Yaskawa INFORM job: TWIN_SKRZYNIA_5140_0_STOPNI_1OBR.JBI

/JOB
//NAME TWIN_SKRZYNIA_5140_0_STOPNI_1OBR
///FOLDERNAME 02-SKRZYNIE_JOBS
//POS
///NPOS 519,519,0,46,4,0
///TOOL 0
///POSTYPE PULSE
///PULSE
C00000=1055,-24125,84372,288,19725,204
C00001=1055,-24125,84372,288,19725,204
C00002=0,-15438,65714,0,-68532,0
C00003=25524,-25821,36823,19654,-58495,38520
C00004=23988,-24960,37134,18595,-57837,38812
C00005=22822,-23954,37534,17811,-57199,39017
C00006=22935,-24057,37491,17887,-57262,38997
C00007=20006,-24258,37408,15644,-56932,39751
C00008=24402,-25289,37013,18874,-58060,38740
C00009=22585,-24665,40358,17164,-59622,30036
C00010=23477,-23257,40205,18030,-58646,29630
C00011=22519,-22398,40568,17384,-58125,29795
C00012=22700,-22567,40495,17506,-58225,29764
C00013=19339,-22794,40398,14955,-57865,30607
C00014=24825,-24328,39798,18931,-59350,29401
C00015=0,-15438,65714,0,-68532,0
C00016=25524,-25821,36823,19654,-58495,38520
C00017=23988,-24960,37134,18595,-57837,38812
C00018=22822,-23954,37534,17811,-57199,39017
C00019=22935,-24057,37491,17887,-57262,38997
C00020=20006,-24258,37408,15644,-56932,39751
C00021=24402,-25289,37013,18874,-58060,38740
C00022=22585,-24665,40358,17164,-59622,30036
C00023=23477,-23257,40205,18030,-58646,29630
C00024=22519,-22398,40568,17384,-58125,29795
C00025=22700,-22567,40495,17506,-58225,29764
C00026=19339,-22794,40398,14955,-57865,30607
C00027=24825,-24328,39798,18931,-59350,29401
C00028=32755,-32613,25711,29640,-48730,33694
C00029=25632,-30899,26166,23992,-46203,35378
C00030=24264,-29862,26497,22996,-45413,35639
C00031=24403,-29974,26459,23097,-45496,35612
C00032=20575,-30233,26374,19602,-44891,36810
C00033=26556,-31526,25988,24663,-46720,35206
C00034=30846,-32795,25752,28021,-48338,30427
C00035=24953,-30697,26306,23444,-45946,31743
C00036=23937,-29910,26558,22702,-45353,31936
C00037=24039,-29993,26530,22778,-45414,31916
C00038=20322,-30240,26449,19379,-44834,33080
C00039=25997,-31433,26093,24205,-46535,31545
C00040=26028,-43665,26580,-39946,8682,24640
C00041=27956,-30595,53065,-101898,6609,54413
C00042=26028,-43663,26580,-39944,8677,24639
C00043=38784,-34544,25404,33956,-51320,34445
C00044=29266,-32676,25756,26732,-47889,36488
C00045=25734,-31262,26119,24020,-46377,37252
C00046=24289,-30200,26441,22967,-45549,37525
C00047=24367,-30262,26420,23025,-45594,37511
C00048=20043,-30544,26331,19080,-44922,38860
C00049=26573,-31816,25967,24631,-46839,37095
C00050=27817,-32566,25782,25532,-47502,36865
C00051=26289,-31635,26016,24424,-46683,37147
C00052=24344,-30243,26427,23007,-45578,37515
C00053=24432,-30312,26405,23072,-45630,37498
C00054=20021,-30599,26315,19050,-44944,38872
C00055=26262,-31616,26021,24405,-46667,37153
C00056=27439,-32346,25835,25259,-47302,36935
C00057=27861,-32554,25785,25570,-47505,36851
C00058=24581,-30384,26384,23190,-45695,37464
C00059=24689,-30466,26358,23269,-45758,37444
C00060=20001,-30771,26264,18999,-45026,38899
C00061=26308,-31607,26026,24448,-46671,37139
C00062=27526,-32360,25834,25329,-47326,36914
C00063=24269,-40076,6479,29767,-34177,34232
C00064=22958,-37632,10123,27061,-35370,35326
C00065=22703,-41294,1722,31272,-29953,33282
C00066=19440,-41515,1663,27208,-29122,34832
C00067=25465,-43501,1200,33269,-31905,32752
C00068=87177,-39066,-1236,81808,-72661,19198
C00069=4794,-34097,38974,4189,-31824,-1302
C00070=4794,-34097,38974,4189,13412,-1302
C00071=11237,-37131,38982,-12694,5333,8253
C00072=6591,-33902,35532,5956,-1761,-1932
C00073=10065,-33530,28876,9373,-31104,-3154
C00074=31877,-32319,25770,29025,-48287,33360
C00075=25178,-31109,26094,23580,-46137,35030
C00076=23652,-29939,26460,22464,-45250,35320
C00077=23742,-30013,26436,22530,-45305,35302
C00078=19630,-30281,26348,18756,-44677,36597
C00079=26056,-31710,25928,24219,-46631,34863
C00080=38095,-40136,7813,41252,-44156,24924
C00081=33231,-38681,8176,37792,-41757,25918
C00082=31538,-37640,8473,36716,-40716,26179
C00083=31687,-37737,8444,36811,-40809,26155
C00084=27389,-38154,8322,32773,-39589,27627
C00085=33834,-39023,8084,38175,-42120,25821
C00086=4801,-35772,25187,4594,-28023,-1125
C00087=-1002,-39861,25115,1795,-37402,-69601
C00088=4264,-34194,25387,4006,-26954,-29436
C00089=4264,-34194,25387,4006,-26954,-81856
C00090=17634,-23800,39238,9573,-31425,-73339
C00091=17837,-27228,32238,10495,-29236,-73805
C00092=17837,-21535,44509,9322,-33342,-73155
C00093=17548,-20734,45666,8935,-33511,-73021
C00094=-20829,-18800,50532,-12466,-37179,-77446
C00095=-20884,-20901,46110,-12960,-35762,-77182
C00096=-20884,-26676,33664,-14451,-31668,-76336
C00097=-20624,-26699,33167,-14265,-31320,-76369
C00098=-33629,-40566,17444,-29603,-33447,-71192
C00099=-33629,-40566,17444,42578,-32312,-84654
C00100=-42160,-31266,16400,42578,-32312,-84654
C00101=-87798,-804,48829,-20188,-26072,-60966
C00102=-76454,-11934,10236,-25964,7954,-64922
C00103=-76448,-11928,10235,-25961,7944,-64914
C00104=-68643,-7759,-23318,-14097,50582,-74897
C00105=-70868,-8793,-8075,-29663,30364,-70765
C00106=-67243,-1968,12282,-49553,26687,-63567
C00107=-68655,-309,14069,-48513,25966,-64203
C00108=-67497,-1678,12591,-49367,26558,-63682
C00109=-71436,-723,2905,-26484,35140,-73726
C00110=-71436,176,6426,-27636,33595,-73066
C00111=-71434,778,8668,-28412,32633,-72624
C00112=-68624,-2689,-85,-28291,36551,-72622
C00113=-99375,3692,5712,40719,48607,-84097
C00114=-94964,4957,10918,40408,44640,-83792
C00115=-93063,6047,12199,39572,43744,-83178
C00116=-94964,4957,10918,40408,44640,-83792
C00117=-94964,5754,13918,41385,43553,-84439
C00118=-94964,4957,10918,40408,44640,-83792
C00119=-90271,-412,-5146,23417,46876,-76529
C00120=-83133,-4088,-8267,6704,41492,-71542
C00121=-83133,-4088,-8267,6704,41492,-71542
C00122=-83133,-4088,-8267,6704,41492,-11598
C00123=-83133,-16026,-8267,6704,41492,-11598
C00124=-83133,-16026,-8267,6704,41492,-11598
C00125=-48225,-19387,30619,3889,32460,-6728
C00126=56943,-39861,25115,1795,-37402,-69601
C00127=29960,-38386,-19607,-115769,-41858,-24264
C00128=65721,-6478,18155,-133323,-22195,3361
C00129=70544,4411,32968,-134868,-18623,4660
C00130=71874,8263,38598,-134556,-17327,4659
C00131=72629,9390,40002,-135279,-16924,5107
C00132=71441,7638,37831,-134139,-17555,4406
C00133=77146,8888,25050,-166574,-32612,18372
C00134=77146,10029,28643,-166204,-31014,18167
C00135=77146,11198,32202,-165803,-29459,17947
C00136=75508,4678,16951,-165715,-35157,17778
C00137=68680,12216,24468,-164340,-40455,-13359
C00138=68362,12845,25743,-164045,-40097,-13561
C00139=68362,13700,28585,-163752,-38808,-13742
C00140=68362,12845,25743,-164045,-40097,-13561
C00141=64993,-1168,28876,-102971,-10760,-49875
C00142=63888,481,30670,-102324,-11438,-50313
C00143=64993,-1168,28876,-102971,-10760,-49875
C00144=58588,-14653,4620,-120782,-19611,-35794
C00145=29960,-38386,-19607,-115769,-41858,-24264
C00146=56943,-39861,25115,1795,-37402,-69601
C00147=-1002,-39861,25115,1795,-37402,-69601
C00148=-1001,-39858,25114,1795,-37402,0
C00149=6591,-33902,35532,5956,-1761,-1932
C00150=6592,-33900,35531,103508,-35512,-26314
C00151=-99253,-13690,44082,59847,13407,-31313
C00152=-85045,-36869,-4353,28502,-22832,-52282
C00153=-92346,-18713,13565,21110,-22545,-55257
C00154=-85370,-14218,16934,32905,-23649,-60330
C00155=-84150,-13282,17685,34842,-23935,-61163
C00156=-82877,-12536,18624,36445,-24482,-61818
C00157=-84150,-13282,17685,34842,-23935,-61163
C00158=-85467,-11480,19558,33086,-23405,-60436
C00159=-84150,-13282,17685,34842,-23935,-61163
C00160=-85732,-21202,11427,30682,-24763,-59235
C00161=-84559,-15616,15722,33768,-24118,-60665
C00162=-84150,-13282,17685,34842,-23935,-61163
C00163=-83260,-12880,18034,36130,-24218,-61709
C00164=-84150,-13282,17685,34842,-23935,-61163
C00165=-85365,-11775,19006,33430,-23307,-60600
C00166=-84150,-13282,17685,34842,-23935,-61163
C00167=-85786,-16909,14677,31743,-23900,-59790
C00168=-84150,-13282,17685,34842,-23935,-61163
C00169=-83215,-12861,18051,36194,-24233,-61735
C00170=-84150,-13282,17685,34842,-23935,-61163
C00171=-85327,-11825,18959,33476,-23327,-60618
C00172=-84150,-13282,17685,34842,-23935,-61163
C00173=-87841,-18519,13420,28367,-23534,-58339
C00174=-84150,-13282,17685,34842,-23935,-61163
C00175=-83292,-12894,18020,36083,-24208,-61688
C00176=-84150,-13282,17685,34842,-23935,-61163
C00177=-85185,-12008,18799,33646,-23400,-60687
C00178=-84150,-13282,17685,34842,-23935,-61163
C00179=-86371,-18277,13606,30568,-23951,-59265
C00180=-84345,-13370,17612,34554,-23873,-61041
C00181=-83240,-12871,18042,36158,-24225,-61720
C00182=-84345,-13370,17612,34554,-23873,-61041
C00183=-85365,-12110,18711,33368,-23345,-60568
C00184=-84345,-13370,17612,34554,-23873,-61041
C00185=-86191,-19647,12567,30467,-24278,-59187
C00186=-84345,-13372,17610,34552,-23873,-61039
C00187=-83096,-12807,18098,36363,-24268,-61804
C00188=-84345,-13372,17610,34552,-23873,-61039
C00189=-85268,-12232,18600,33480,-23393,-60612
C00190=-84345,-13372,17610,34552,-23873,-61039
C00191=-84814,-16043,15376,33312,-24093,-60464
C00192=-84104,-13265,17702,34906,-23948,-61189
C00193=-82960,-12743,18153,36555,-24313,-61887
C00194=-84104,-13265,17702,34906,-23948,-61189
C00195=-84979,-12194,18635,33901,-23496,-60788
C00196=-84104,-13265,17702,34906,-23948,-61189
C00197=-86610,-16845,14732,30573,-23614,-59301
C00198=-84104,-13265,17702,34906,-23948,-61189
C00199=-82793,-12667,18222,36790,-24370,-61986
C00200=-84104,-13265,17702,34906,-23948,-61189
C00201=-84888,-12305,18537,34004,-23540,-60830
C00202=-84104,-13265,17702,34906,-23948,-61189
C00203=-83806,-19585,12613,33764,-25080,-60559
C00204=-83675,-13072,17868,35530,-24083,-61453
C00205=-82553,-12556,18319,37130,-24451,-62127
C00206=-83675,-13072,17868,35530,-24083,-61453
C00207=-84378,-12223,18610,34735,-23716,-61138
C00208=-83675,-13072,17868,35530,-24083,-61453
C00209=-87149,-17993,13826,29513,-23647,-58830
C00210=-84104,-13265,17702,34906,-23948,-61189
C00211=-82640,-12594,18285,37014,-24425,-62079
C00212=-84104,-13265,17702,34906,-23948,-61189
C00213=-84792,-12429,18430,34119,-23592,-60877
C00214=-84104,-13265,17702,34906,-23948,-61189
C00215=-83583,-9185,30892,23668,-36042,-57025
C00216=-85789,-8328,35795,20592,-37093,-55378
C00217=-85786,-16735,14816,31782,-23869,-59812
C00218=-84103,-13263,17702,34906,-23947,-61191
C00219=-83225,-12865,18046,36177,-24227,-61729
C00220=-84103,-13263,17702,34906,-23947,-61191
C00221=-84774,-12447,18412,34138,-23599,-60886
C00222=-84103,-13263,17702,34906,-23947,-61191
C00223=-86149,-16246,6730,18897,-35239,-57128
C00224=-86244,-15289,7532,18875,-35060,-57127
C00225=-85361,-14893,7870,19824,-35193,-57574
C00226=-86244,-15289,7532,18875,-35060,-57127
C00227=-86889,-14409,8282,18264,-34784,-56850
C00228=-86244,-15289,7532,18875,-35060,-57127
C00229=-90262,-21765,2389,14114,-35574,-54847
C00230=-90262,-21765,2389,28730,-17672,-54847
C00231=-89967,-19086,25635,28730,-17672,-54847
C00232=568,-24029,84339,168,19981,112
C00233=568,-24677,83015,164,20405,113
C00234=101153,-24598,83176,165,20353,113
C00235=101153,-24598,83176,165,20353,113
C00236=89967,-19086,25635,-28730,-17672,54847
C00237=90262,-21765,2389,-28730,-17672,54847
C00238=86932,-18662,4771,-17876,-35519,56628
C00239=86578,-15436,7408,-18515,-35011,56957
C00240=85428,-14922,7844,-19753,-35183,57541
C00241=84405,-14447,8250,-20842,-35348,58054
C00242=85428,-14922,7844,-19753,-35183,57541
C00243=86134,-13973,8661,-19091,-34881,57237
C00244=85428,-14922,7844,-19753,-35183,57541
C00245=85786,-16735,14816,-31782,-23869,59812
C00246=83514,-12996,17929,-35760,-24132,61552
C00247=82296,-12429,18424,-37488,-24534,62281
C00248=83514,-12996,17929,-35760,-24132,61552
C00249=84266,-12085,18725,-34910,-23738,61214
C00250=83514,-12996,17929,-35760,-24132,61552
C00251=87323,-6914,39851,-18853,-38149,44508
C00252=83118,-12818,18089,-36330,-24263,61791
C00253=81969,-12276,18566,-37944,-24648,62472
C00254=83118,-12818,18089,-36330,-24263,61791
C00255=83927,-11846,18941,-35423,-23842,61433
C00256=83118,-12818,18089,-36330,-24263,61791
C00257=83806,-19585,12613,-33764,-25080,60559
C00258=83148,-12832,18077,-36287,-24254,61773
C00259=81889,-12236,18598,-38058,-24676,62520
C00260=83148,-12832,18077,-36287,-24254,61773
C00261=83900,-11930,18867,-35446,-23862,61440
C00262=83148,-12832,18077,-36287,-24254,61773
C00263=86610,-16845,14732,-30573,-23614,59301
C00264=82493,-13239,17725,-37070,-24559,62089
C00265=81442,-12739,18159,-38529,-24915,62703
C00266=82493,-13239,17725,-37070,-24559,62089
C00267=83435,-12133,18689,-36040,-24063,61682
C00268=82493,-13239,17725,-37070,-24559,62089
C00269=84814,-16043,15376,-33312,-24093,60464
C00270=82555,-13613,17404,-36910,-24580,62015
C00271=81369,-13053,17885,-38558,-24979,62709
C00272=82555,-13613,17404,-36910,-24580,62015
C00273=83568,-12431,18429,-35805,-24046,61580
C00274=82555,-13613,17404,-36910,-24580,62015
C00275=86191,-19647,12567,-30467,-24278,59187
C00276=82500,-13648,17375,-36975,-24607,62039
C00277=81594,-13224,17740,-38236,-24911,62571
C00278=82500,-13648,17375,-36975,-24607,62039
C00279=83449,-12543,18332,-35941,-24104,61633
C00280=82500,-13648,17375,-36975,-24607,62039
C00281=86371,-18277,13606,-30568,-23951,59265
C00282=82904,-13790,17251,-36416,-24470,61808
C00283=81796,-13275,17692,-37971,-24838,62464
C00284=82904,-13790,17251,-36416,-24470,61808
C00285=83696,-12867,18046,-35547,-24051,61466
C00286=82904,-13790,17251,-36416,-24470,61808
C00287=87841,-18519,13420,-28367,-23534,58339
C00288=82748,-13879,17174,-36603,-24542,61883
C00289=81789,-13434,17554,-37946,-24861,62449
C00290=82748,-13879,17174,-36603,-24542,61883
C00291=83603,-12888,18026,-35668,-24086,61514
C00292=82748,-13879,17174,-36603,-24542,61883
C00293=85786,-16909,14677,-31743,-23900,59790
C00294=82339,-14116,16972,-37087,-24733,62079
C00295=81557,-13752,17280,-38171,-24994,62536
C00296=82339,-14116,16972,-37087,-24733,62079
C00297=83390,-12909,18006,-35951,-24172,61633
C00298=82339,-14116,16972,-37087,-24733,62079
C00299=85732,-21202,11427,-30682,-24763,59235
C00300=82398,-14365,16763,-36952,-24745,62014
C00301=81340,-13876,17176,-38416,-25096,62632
C00302=82398,-14365,16763,-36952,-24745,62014
C00303=83629,-12951,17972,-35620,-24090,61491
C00304=82398,-14365,16763,-36952,-24745,62014
C00305=92346,-18713,13565,-21110,-22545,55257
C00306=82794,-13980,17083,-36511,-24538,61844
C00307=81697,-13472,17516,-38043,-24902,62488
C00308=82794,-13980,17083,-36511,-24538,61844
C00309=83767,-12847,18056,-35444,-24023,61424
C00310=82794,-13980,17083,-36511,-24538,61844
C00311=85045,-36869,-4353,-28502,-22832,52282
C00312=69856,-53931,-13446,-33557,-28911,29591
C00313=73943,-28815,39553,-16801,-45089,19004
C00314=0,-24029,84339,0,19981,0
C00315=0,-24029,84339,0,19981,0
C00316=0,-52280,40443,0,6876,0
C00317=63961,-36661,14391,66570,-58199,13439
C00318=49610,-38907,493,64064,-47684,11073
C00319=46995,-37828,887,63047,-46050,11165
C00320=46896,-37872,871,62973,-46008,11193
C00321=54160,-39955,137,66075,-50361,10746
C00322=0,-52280,40443,0,6876,0
C00323=0,-52280,40443,0,6876,0
C00324=42978,-45587,7631,48214,-41849,18034
C00325=36694,-44945,-1657,49443,-34807,15750
C00326=45692,-38977,-3583,70505,-41697,11397
C00327=45346,-39151,-3505,69979,-41499,11612
C00328=45286,-39124,-3496,69961,-41460,11611
C00329=34756,-41823,-6138,63561,-31389,22119
C00330=59828,-44646,-5405,72855,-48572,12139
C00331=0,-38761,66314,0,-763,0
C00332=0,-44757,54667,0,2744,0
C00333=40382,-38226,12225,48505,-40693,16039
C00334=55481,-27484,23768,62968,-54833,11978
C00335=49932,-26591,24189,59970,-51981,12550
C00336=49523,-31326,12269,55024,-55929,13117
C00337=55330,-33748,11238,57660,-59334,12681
C00338=78664,-24436,10378,82837,-79111,12029
C00339=75189,-23065,11287,81851,-76948,11927
C00340=75189,-45249,11287,81851,-38847,11927
C00341=29880,-45249,11287,43145,-11324,11927
C00342=0,-24029,84339,0,19981,0
C00343=0,-24026,84338,1,19977,2
C00344=4264,-34194,25387,4006,-26954,-29436
C00345=4264,-34194,25387,4006,-26954,-81856
C00346=18580,-28601,30698,11472,-29284,-74138
C00347=-23778,-26243,38799,-16502,-35132,-75964
C00348=18580,-28601,30698,11472,-29284,-74138
C00349=4264,-34194,25387,4006,-26954,-81856
C00350=4264,-34194,25387,4006,-26954,-29436
C00351=1,-24024,84337,2,19973,1
C00352=-64243,-26178,31107,-39513,40312,-5844
C00353=-72148,3973,56008,-35470,42045,-10522
C00354=-72090,16396,76301,-42067,35650,-6519
C00355=-69388,15725,61378,-31740,35177,-8719
C00356=-69127,27099,75569,-32744,34250,-8088
C00357=-67573,2495,11285,-21767,57629,-15193
C00358=-77819,19629,29798,-10454,63174,-20704
C00359=-72990,23583,14304,-10735,77209,-20379
C00360=-74593,38003,46707,-11043,65751,-19814
C00361=-73236,38943,48295,-11400,65557,-19316
C00362=-73329,42107,51779,-6346,67443,-19636
C00363=-87142,34654,46174,17622,63862,-25393
C00364=-87240,36727,48611,18897,66604,-25032
C00365=-99033,21517,12213,24947,79702,-26203
C00366=-91500,-14196,-34781,24472,81625,-22832
C00367=-100472,-45007,-27818,8167,67201,-29302
C00368=0,-36642,16905,0,48372,0
C00369=66009,-61997,-62105,21406,63483,18379
C00370=97242,-23579,-39442,10179,68876,30321
C00371=73684,-7073,-17511,24638,68131,29022
C00372=59136,7235,6676,33270,66602,27507
C00373=54816,14937,6234,39741,69494,31070
C00374=54365,20668,19279,41017,66202,29418
C00375=64503,4223,2857,29650,48528,26647
C00376=75622,3202,-3149,3890,49494,34281
C00377=88036,13177,2413,-18568,66573,35876
C00378=90462,21593,10123,-22613,76266,34479
C00379=92450,29224,20002,-25750,81642,33727
C00380=94949,8131,-12163,-20291,74229,36861
C00381=94949,8084,-13484,-20215,75047,36712
C00382=70412,-34016,-52305,-11724,65624,29757
C00383=44268,-30306,-1568,-7370,48673,18708
C00384=1,-24024,84337,2,19973,1
C00385=1,-24024,84337,2,19973,1
C00386=3796,-57671,22373,2336,-25309,-753
C00387=52632,-34554,16626,51161,-63050,5622
C00388=59461,-32779,9832,66317,-58406,17312
C00389=52359,-27861,19114,60105,-56373,14901
C00390=51089,-17517,41583,51411,-64544,19432
C00391=62932,-33588,12189,66848,-61063,18031
C00392=55769,-31640,17107,64026,-54372,11197
C00393=49968,-26926,23568,59773,-52215,12586
C00394=49609,-31413,12230,55051,-55993,13121
C00395=55330,-33748,11238,57660,-59334,12681
C00396=62932,-33588,12189,66848,-61063,18031
C00397=1,-24024,84337,2,19973,1
C00398=1,-24024,84337,2,19973,1
C00399=57188,-41777,19973,48132,-58706,4905
C00400=55566,-48748,-16991,79805,-45048,-6941
C00401=49908,-48716,-25784,90749,-41340,-3650
C00402=44463,-47168,-25441,90895,-37884,-4475
C00403=44064,-46950,-25361,90973,-37634,-4568
C00404=55479,-50244,-26473,91085,-44870,-3042
C00405=12119,-24859,71505,13236,4440,2633
C00406=-91085,-34291,10385,1908,-24348,-42097
C00407=-86191,-19647,12567,30467,-24278,-59187
C00408=-99260,-11699,19072,-14181,-20214,-40097
C00409=-98334,-11556,19569,-10380,-20328,-41527
C00410=-99474,-20389,12397,-11593,-22150,-41069
C00411=0,-52280,40443,0,6876,0
C00412=85348,-24204,23536,-13963,-15515,44275
C00413=84670,-17015,14597,-33277,-24304,60423
C00414=97099,-12623,18260,8611,-19973,42508
C00415=97182,-12918,18001,8747,-20027,42449
C00416=96230,-24528,9149,6144,-22576,43630
C00417=0,-52280,40443,0,6876,0
C00418=0,-52280,40443,0,6876,0
C00419=-90140,-60305,18108,-2708,1721,-7625
C00420=-95594,-27428,6866,-4663,-19832,-42154
C00421=-99356,-13410,18355,-15385,-17730,-37479
C00422=-99405,-10878,20508,-15853,-17333,-37255
C00423=-99155,-10757,20617,-15328,-17277,-37477
C00424=-99152,-3438,39174,-10973,-24351,-39660
C00425=-99136,-3399,39184,-10956,-24327,-39665
C00426=-100183,-18601,14070,-16273,-18800,-37146
C00427=-90140,-60305,18108,-2708,1721,-7625
C00428=0,-52280,40443,0,6876,0
C00429=84259,-57935,27522,-3761,3673,6310
C00430=86507,-39672,4297,-27618,-16640,46340
C00431=70477,-27878,7073,-45786,-32339,64941
C00432=84043,-16293,15174,-34312,-24409,60872
C00433=82317,-21832,-7005,-55296,-17985,71248
C00434=99154,-17369,4403,32227,-9753,28926
C00435=99154,-17369,4403,32227,-9753,28926
C00436=98946,-17182,4556,31649,-9649,29182
C00437=100388,-17987,13832,15751,-21517,39479
C00438=86507,-39672,4297,-27618,-16640,46340
C00439=84259,-57935,27522,-3761,3673,6310
C00440=0,-52280,40443,0,6876,0
C00441=0,-27933,77061,0,20812,0
C00442=0,-27933,77061,0,20812,0
C00443=0,-52280,40443,0,6876,0
C00444=-91970,-60791,14435,-3343,512,-9412
C00445=-99196,-15868,16098,-13748,-19297,-38710
C00446=-99196,-15868,16098,-13748,-19297,-38710
C00447=-99196,-15868,16098,-13748,-19297,-38710
C00448=-85815,-11758,19597,31748,-21097,-58265
C00449=-87383,-11883,19487,26986,-20206,-56250
C00450=-99562,-16264,15781,-14410,-19427,-38431
C00451=-99196,-15868,16098,-13748,-19297,-38710
C00452=-91970,-60791,14435,-3343,512,-9412
C00453=0,-52280,40443,0,6876,0
C00454=91083,-60784,14823,-9043,-825,15173
C00455=83869,-19403,12921,-33769,-24740,60260
C00456=83869,-19403,12921,-33769,-24740,60260
C00457=83420,-14897,16486,-35538,-24144,61113
C00458=90568,-11796,19695,-13982,-20788,51525
C00459=90396,-11649,19890,-14205,-20868,51587
C00460=95871,-14889,15992,4901,-19605,43825
C00461=83869,-19403,12921,-33769,-24740,60260
C00462=91083,-60784,14823,-9043,-825,15173
C00463=0,-52280,40443,0,6876,0
C00464=-91526,-60598,16699,7584,176,-13289
C00465=-94392,-6553,48683,5805,-47321,-49764
C00466=-88951,-345,54953,10686,-47392,-51569
C00467=-88172,5833,62122,11322,-47753,-51785
C00468=-90970,-13982,9528,8812,-34392,-51924
C00469=-84917,-15593,15742,33275,-23984,-60461
C00470=-81669,-15982,15425,37506,-25258,-62202
C00471=-79867,-25377,9541,37586,-25936,-59971
C00472=-91415,-60262,16631,7870,-73,-13734
C00473=24,-24029,84339,7,19981,5
C00474=160,-24029,84339,47,19981,32
C00475=99096,-24029,84339,47,19981,32
C00476=99096,-24029,84339,47,19981,32
C00477=89967,-19086,25635,-28730,-17672,54847
C00478=85786,-16735,14816,-31782,-23869,59812
C00479=83492,-14473,16674,-35480,-24338,61406
C00480=82750,-11489,19288,-37313,-24360,62208
C00481=85452,-13705,8809,-19525,-34825,57501
C00482=85505,-16299,6686,-19564,-35388,57437
C00483=89967,-19086,25635,-28730,-17672,54847
C00484=568,-24029,84339,168,19981,112
C00485=568,-24029,84339,168,19981,112
C00486=-91970,-60791,14435,-3343,512,-9412
C00487=-86948,-23217,10819,28314,-23349,-56438
C00488=-85895,-16522,15767,31843,-22281,-58087
C00489=-93602,1725,52992,2981,-38211,-34794
C00490=-93409,-737,47229,3345,-36106,-34967
C00491=-86145,-24679,9854,29028,-23971,-56682
C00492=-100471,-58311,4157,14142,-4822,-27614
C00493=-68517,-58311,4157,14142,-4822,-27614
C00494=0,-52280,40443,0,6876,0
C00495=91083,-60784,14823,-9043,-825,15173
C00496=83869,-19403,12921,-33769,-24740,60260
C00497=82620,-18743,14708,-32942,-26226,58979
C00498=83365,-11429,20745,-33501,-24845,59379
C00499=83361,-11160,20982,-33549,-24816,59402
C00500=84798,-22668,11879,-29033,-26372,57255
C00501=91083,-60784,14823,-9043,-825,15173
C00502=0,-52280,40443,0,6876,0
C00503=-6369,-39206,65423,-4801,-482,2563
C00504=-97287,-29142,12714,-8673,-22288,-37832
C00505=-86191,-19647,12567,30467,-24278,-59187
C00506=-85671,-16302,15857,30808,-24404,-58999
C00507=-100033,-10430,22389,-14713,-22552,-38787
C00508=-95758,-10871,21797,-1120,-21702,-44724
C00509=-87910,-17792,15835,25414,-24996,-56048
C00510=-97287,-29142,12714,-8673,-22288,-37832
C00511=0,-52280,40443,0,6876,0
C00512=92301,-25634,22749,2368,-15645,37646
C00513=83738,-18329,13570,-34202,-24868,60772
C00514=90096,-13099,18146,-15422,-20883,52700
C00515=93330,-13245,17928,-4627,-20146,48105
C00516=80226,-20465,12178,-39626,-27411,62762
C00517=92301,-25634,22749,2368,-15645,37646
C00518=0,-52280,40443,0,6876,0
BC00000=413138
BC00001=413138
BC00002=413138
BC00003=290246
BC00004=290246
BC00005=290246
BC00006=290246
BC00007=290246
BC00008=290246
BC00009=347127
BC00010=347132
BC00011=347132
BC00012=347132
BC00013=347132
BC00014=347132
BC00015=413138
BC00016=413134
BC00017=413134
BC00018=413134
BC00019=413134
BC00020=413134
BC00021=413134
BC00022=474623
BC00023=474628
BC00024=474628
BC00025=474628
BC00026=474628
BC00027=474628
BC00028=522849
BC00029=522849
BC00030=522849
BC00031=522849
BC00032=522849
BC00033=522849
BC00034=586045
BC00035=586045
BC00036=586045
BC00037=586045
BC00038=586045
BC00039=586045
BC00040=479622
BC00041=618860
BC00042=673957
BC00043=655410
BC00044=655410
BC00045=655410
BC00046=655410
BC00047=655410
BC00048=655410
BC00049=655410
BC00050=708270
BC00051=708270
BC00052=708270
BC00053=708270
BC00054=708270
BC00055=708270
BC00056=770184
BC00057=770184
BC00058=770184
BC00059=770184
BC00060=770184
BC00061=770184
BC00062=823730
BC00063=829967
BC00064=829969
BC00065=829970
BC00066=829970
BC00067=829970
BC00068=838761
BC00069=740349
BC00070=687700
BC00071=771943
BC00072=861898
BC00073=881669
BC00074=901229
BC00075=901229
BC00076=901229
BC00077=901229
BC00078=901229
BC00079=901229
BC00080=949836
BC00081=949836
BC00082=949836
BC00083=949836
BC00084=949836
BC00085=949836
BC00086=922151
BC00087=915598
BC00088=911152
BC00089=906014
BC00090=926513
BC00091=926513
BC00092=930959
BC00093=930959
BC00094=930959
BC00095=930959
BC00096=930959
BC00097=930959
BC00098=930959
BC00099=930959
BC00100=930959
BC00101=930959
BC00102=930959
BC00103=948711
BC00104=959797
BC00105=976501
BC00106=976501
BC00107=976501
BC00108=976501
BC00109=976501
BC00110=976501
BC00111=976502
BC00112=976502
BC00113=976502
BC00114=976502
BC00115=976502
BC00116=976502
BC00117=976502
BC00118=976502
BC00119=966879
BC00120=952245
BC00121=926980
BC00122=926980
BC00123=926980
BC00124=893798
BC00125=874726
BC00126=930959
BC00127=930959
BC00128=930959
BC00129=947173
BC00130=952334
BC00131=952334
BC00132=952334
BC00133=952334
BC00134=952334
BC00135=952334
BC00136=952334
BC00137=952334
BC00138=952334
BC00139=952334
BC00140=952334
BC00141=952334
BC00142=952334
BC00143=952334
BC00144=946821
BC00145=930959
BC00146=900237
BC00147=900237
BC00148=930961
BC00149=861898
BC00150=861901
BC00151=861901
BC00152=931504
BC00153=960562
BC00154=960559
BC00155=960559
BC00156=960559
BC00157=960559
BC00158=960559
BC00159=960559
BC00160=902188
BC00161=902188
BC00162=902188
BC00163=902188
BC00164=902188
BC00165=902188
BC00166=902188
BC00167=840744
BC00168=840744
BC00169=840744
BC00170=840744
BC00171=840744
BC00172=840744
BC00173=779300
BC00174=779300
BC00175=779300
BC00176=779300
BC00177=779300
BC00178=779300
BC00179=717855
BC00180=717855
BC00181=717855
BC00182=717855
BC00183=717855
BC00184=717855
BC00185=656405
BC00186=656405
BC00187=656405
BC00188=656405
BC00189=656405
BC00190=656405
BC00191=594961
BC00192=594961
BC00193=594961
BC00194=594961
BC00195=594961
BC00196=594961
BC00197=533517
BC00198=533517
BC00199=533517
BC00200=533517
BC00201=533517
BC00202=533517
BC00203=472073
BC00204=472073
BC00205=472073
BC00206=472073
BC00207=472073
BC00208=472073
BC00209=410629
BC00210=410629
BC00211=410629
BC00212=410629
BC00213=410629
BC00214=410629
BC00215=410629
BC00216=349186
BC00217=349186
BC00218=349186
BC00219=349186
BC00220=349186
BC00221=349186
BC00222=349186
BC00223=336469
BC00224=336469
BC00225=336469
BC00226=336469
BC00227=336469
BC00228=336469
BC00229=336469
BC00230=336469
BC00231=336469
BC00232=336469
BC00233=511557
BC00234=512005
BC00235=363797
BC00236=336469
BC00237=336469
BC00238=337415
BC00239=337415
BC00240=337415
BC00241=337415
BC00242=337415
BC00243=337415
BC00244=337415
BC00245=349186
BC00246=350137
BC00247=350137
BC00248=350137
BC00249=350137
BC00250=350137
BC00251=410629
BC00252=411580
BC00253=411580
BC00254=411580
BC00255=411580
BC00256=411580
BC00257=472073
BC00258=473025
BC00259=473025
BC00260=473025
BC00261=473025
BC00262=473025
BC00263=533517
BC00264=534468
BC00265=534468
BC00266=534468
BC00267=534468
BC00268=534468
BC00269=594961
BC00270=594961
BC00271=594961
BC00272=594961
BC00273=594961
BC00274=594961
BC00275=656405
BC00276=657350
BC00277=657350
BC00278=657350
BC00279=657350
BC00280=657350
BC00281=717855
BC00282=718799
BC00283=718799
BC00284=718799
BC00285=718799
BC00286=718799
BC00287=779300
BC00288=780245
BC00289=780245
BC00290=780245
BC00291=780245
BC00292=780245
BC00293=840744
BC00294=841691
BC00295=841691
BC00296=841691
BC00297=841691
BC00298=841691
BC00299=902188
BC00300=903136
BC00301=903136
BC00302=903136
BC00303=903136
BC00304=903136
BC00305=963634
BC00306=963633
BC00307=963633
BC00308=963633
BC00309=963633
BC00310=963633
BC00311=931504
BC00312=861901
BC00313=861901
BC00314=769966
BC00315=769966
BC00316=716865
BC00317=660977
BC00318=660977
BC00319=660977
BC00320=717171
BC00321=717171
BC00322=716865
BC00323=796033
BC00324=895097
BC00325=895097
BC00326=895097
BC00327=945882
BC00328=959029
BC00329=966042
BC00330=945882
BC00331=840120
BC00332=538973
BC00333=485226
BC00334=456696
BC00335=456696
BC00336=417276
BC00337=417276
BC00338=493986
BC00339=514306
BC00340=514306
BC00341=514306
BC00342=493986
BC00343=797003
BC00344=895791
BC00345=895791
BC00346=895791
BC00347=900237
BC00348=895791
BC00349=895791
BC00350=895791
BC00351=797001
BC00352=812363
BC00353=812363
BC00354=853712
BC00355=873598
BC00356=898537
BC00357=930469
BC00358=930469
BC00359=957978
BC00360=957978
BC00361=957978
BC00362=957979
BC00363=957979
BC00364=957980
BC00365=957980
BC00366=957980
BC00367=872638
BC00368=831236
BC00369=914776
BC00370=953896
BC00371=953897
BC00372=953897
BC00373=984144
BC00374=984144
BC00375=984144
BC00376=984144
BC00377=984144
BC00378=984147
BC00379=984147
BC00380=984147
BC00381=957741
BC00382=957741
BC00383=888928
BC00384=797001
BC00385=461290
BC00386=507200
BC00387=551170
BC00388=578587
BC00389=593948
BC00390=529848
BC00391=529848
BC00392=333808
BC00393=332068
BC00394=295166
BC00395=294388
BC00396=529848
BC00397=461290
BC00398=663315
BC00399=778314
BC00400=778312
BC00401=778312
BC00402=778312
BC00403=838222
BC00404=838222
BC00405=566410
BC00406=679663
BC00407=656405
BC00408=656405
BC00409=717855
BC00410=717855
BC00411=717855
BC00412=662303
BC00413=657350
BC00414=657350
BC00415=718803
BC00416=718803
BC00417=717855
BC00418=792672
BC00419=792672
BC00420=896850
BC00421=895720
BC00422=895720
BC00423=957178
BC00424=957178
BC00425=959216
BC00426=957178
BC00427=792672
BC00428=792672
BC00429=792672
BC00430=887446
BC00431=903126
BC00432=903126
BC00433=923336
BC00434=964577
BC00435=976097
BC00436=978451
BC00437=964577
BC00438=887446
BC00439=792672
BC00440=792672
BC00441=700249
BC00442=546214
BC00443=546214
BC00444=546211
BC00445=546211
BC00446=406776
BC00447=406776
BC00448=406778
BC00449=468200
BC00450=468200
BC00451=546211
BC00452=546211
BC00453=546214
BC00454=546214
BC00455=507604
BC00456=410782
BC00457=410782
BC00458=410782
BC00459=472720
BC00460=472720
BC00461=507604
BC00462=546214
BC00463=546214
BC00464=516757
BC00465=383716
BC00466=349186
BC00467=349186
BC00468=336469
BC00469=349186
BC00470=410629
BC00471=416512
BC00472=515801
BC00473=520018
BC00474=474013
BC00475=474013
BC00476=403108
BC00477=336469
BC00478=349186
BC00479=349186
BC00480=349186
BC00481=337415
BC00482=337415
BC00483=336469
BC00484=336469
BC00485=428401
BC00486=546211
BC00487=591088
BC00488=591088
BC00489=591088
BC00490=531116
BC00491=529640
BC00492=529640
BC00493=529640
BC00494=529640
BC00495=546214
BC00496=589919
BC00497=595627
BC00498=595627
BC00499=534177
BC00500=534177
BC00501=546214
BC00502=529640
BC00503=651195
BC00504=765890
BC00505=777968
BC00506=778453
BC00507=779252
BC00508=840748
BC00509=840748
BC00510=765890
BC00511=717855
BC00512=741100
BC00513=780224
BC00514=780222
BC00515=841743
BC00516=841743
BC00517=741100
BC00518=717855
///POSTYPE BASE
///RECTAN
///RCONF 1,0,0,0,0,0,0,0,0,0,0,0,0,0,0,0,0,0,0,0,0,0,0,0
P00006=0.000,0.000,0.000,0.0000,0.0000,0.0000
P00098=-0.089,-2.467,4.059,0.0000,0.0000,0.0000
P00099=0.011,-2.380,1.226,0.0000,0.0000,0.0000
P00100=-0.081,2.558,4.482,0.0000,0.0000,0.0000
P00101=0.030,-2.286,2.993,0.0000,0.0000,0.0000
P00102=-0.005,-1.108,1.644,0.0000,0.0000,0.0000
P00103=-0.094,-3.400,4.200,0.0000,0.0000,0.0000
P00104=0.043,-2.127,5.826,0.0000,0.0000,0.0000
P00105=-0.043,0.662,5.286,0.0000,0.0000,0.0000
P00106=-0.018,-2.519,0.237,0.0000,0.0000,0.0000
P00107=-0.008,-4.537,-4.500,0.0000,0.0000,0.0000
P00108=0.014,-3.040,2.637,0.0000,0.0000,0.0000
P00109=0.017,-3.622,2.341,0.0000,0.0000,0.0000
P00110=7346.140,158.997,-946.107,-0.1876,37.7131,-155.1643
P00111=7345.905,-141.160,-945.062,8.1413,34.2244,-174.1788
P00112=7393.287,158.977,-939.640,-0.1938,37.7128,-155.1905
P00113=7393.259,-141.170,-939.228,8.1507,34.2195,-174.1496
///RCONF 0,0,0,0,0,0,0,0,0,0,0,0,0,0,0,0,0,0,0,0,0,0,0,0
P00280=-0.761,-1.221,0.004,0.0000,0.0000,0.0000
///RCONF 1,0,0,0,0,0,0,0,0,0,0,0,0,0,0,0,0,0,0,0,0,0,0,0
P00281=-0.866,-3.587,-0.008,0.0000,0.0000,0.0000
///RCONF 0,0,0,0,1,0,0,0,0,0,0,0,0,0,0,0,0,0,0,0,0,0,0,0
P00290=-0.023,-0.050,5.560,0.0000,0.0000,0.0000
///RCONF 1,0,0,0,0,0,0,0,0,0,0,0,0,0,0,0,0,0,0,0,0,0,0,0
P00291=0.002,-0.893,4.526,0.0000,0.0000,0.0000
P00300=-0.036,-1.505,2.318,0.0000,0.0000,0.0000
P00301=0.046,-2.112,7.779,0.0000,0.0000,0.0000
P00302=-0.180,-2.409,6.326,0.0000,0.0000,0.0000
///RCONF 0,0,0,0,0,0,0,0,0,0,0,0,0,0,0,0,0,0,0,0,0,0,0,0
P00303=-0.004,-1.437,-4.584,0.0000,0.0000,0.0000
P00304=0.028,-1.666,-4.234,0.0000,0.0000,0.0000
P00305=-0.003,-1.920,-3.501,0.0000,0.0000,0.0000
P00306=0.015,-2.252,-3.054,0.0000,0.0000,0.0000
P00307=0.019,-2.151,-5.077,0.0000,0.0000,0.0000
P00308=-0.003,-2.092,-4.888,0.0000,0.0000,0.0000
P00309=-0.040,-2.205,-4.992,0.0000,0.0000,0.0000
P00310=-0.006,-2.490,-5.925,0.0000,0.0000,0.0000
P00311=-0.007,-2.079,-5.307,0.0000,0.0000,0.0000
P00350=11.519,-0.008,1.149,0.0000,0.0000,0.0000
P00351=13.563,-0.027,-0.653,0.0000,0.0000,0.0000
P00352=13.252,-0.027,-0.827,0.0000,0.0000,0.0000
P00353=10.971,-0.082,0.776,0.0000,0.0000,0.0000
P00354=-0.024,2.508,-1.824,0.0000,0.0000,0.0000
P00355=-0.001,2.528,-1.131,0.0000,0.0000,0.0000
P00356=-0.034,2.921,-0.262,0.0000,0.0000,0.0000
P00357=0.003,3.386,-0.091,0.0000,0.0000,0.0000
P00358=0.014,3.037,-0.020,0.0000,0.0000,0.0000
P00359=-0.005,2.731,0.912,0.0000,0.0000,0.0000
P00360=-0.011,3.412,0.438,0.0000,0.0000,0.0000
P00361=0.018,3.050,1.253,0.0000,0.0000,0.0000
P00777=-1.000,0.000,-1.000,0.0000,0.0000,0.0000
BP00110=5931.608
BP00111=5960.552
BP00112=5960.545
BP00113=5960.552
//INST
///DATE 2024/12/18 10:28
///ATTR SC,RW
///GROUP1 RB1,BS1
NOP
CALL JOB:MOVE_INTO_TUNNEL
MOVJ C00000 BC00000 VJ=30.00
'------------------------
'------------------------
'SPOINA SRODEK DOL
'------------------------
'------------------------
'POMIAR DO WYJ!! PRZEROBIC NA STD
MOVJ C00001 BC00001 VJ=40.00
MOVJ C00002 BC00002 VJ=40.00
'SPOINA_PODLOGA_BRAK_ROZP
MOVJ C00003 BC00003 VJ=20.00 PL=0
MOVL C00004 BC00004 V=166.7 PL=0
REFP 3 C00005 BC00005
CALL JOB:SEARCH-R1
SET P0098 P0006
SFTON P0098
MOVL C00006 BC00006 V=66.7 PL=0
REFP 3 C00007 BC00007
CALL JOB:SEARCH-R1
SET P0098 P0006
SFTON P0098
MOVL C00008 BC00008 V=333.3 PL=0
SFTOF
'W3L
MOVL C00009 BC00009 V=666.7
MOVL C00010 BC00010 V=166.7 PL=0
REFP 3 C00011 BC00011
CALL JOB:SEARCH-R1
SET P0099 P0006
SFTON P0099
MOVL C00012 BC00012 V=166.7 PL=0
REFP 3 C00013 BC00013
CALL JOB:SEARCH-R1
SET P0099 P0006
SFTON P0099
MOVL C00014 BC00014 V=333.3 PL=0
SFTOF
'SPOINA_PODLOGA_BRAK_ROZP
MOVJ C00015 BC00015 VJ=40.00
'W3P
MOVJ C00016 BC00016 VJ=20.00 PL=0
MOVL C00017 BC00017 V=166.7 PL=0
REFP 3 C00018 BC00018
CALL JOB:SEARCH-R1
SET P0100 P0006
SFTON P0100
MOVL C00019 BC00019 V=66.7 PL=0
REFP 3 C00020 BC00020
CALL JOB:SEARCH-R1
SET P0100 P0006
SFTON P0100
MOVL C00021 BC00021 V=333.3 PL=0
SFTOF
'W3L
MOVL C00022 BC00022 V=666.7
MOVL C00023 BC00023 V=166.7 PL=0
REFP 3 C00024 BC00024
CALL JOB:SEARCH-R1
SET P0101 P0006
SFTON P0101
MOVL C00025 BC00025 V=166.7 PL=0
REFP 3 C00026 BC00026
CALL JOB:SEARCH-R1
SET P0101 P0006
SFTON P0101
MOVL C00027 BC00027 V=333.3 PL=0
SFTOF
'W9P
MOVL C00028 BC00028 V=666.7
MOVL C00029 BC00029 V=166.7
REFP 3 C00030 BC00030
CALL JOB:SEARCH-R1
SET P0102 P0006
SFTON P0102
MOVL C00031 BC00031 V=166.7 PL=0
REFP 3 C00032 BC00032
CALL JOB:SEARCH-R1
SET P0102 P0006
SFTON P0102
MOVL C00033 BC00033 V=333.3 PL=0
'W9L
MOVL C00034 BC00034 V=666.7
MOVL C00035 BC00035 V=166.7
REFP 3 C00036 BC00036
CALL JOB:SEARCH-R1
SET P0103 P0006
SFTON P0103
MOVL C00037 BC00037 V=166.7 PL=0
REFP 3 C00038 BC00038
CALL JOB:SEARCH-R1
SET P0103 P0006
SFTON P0103
MOVL C00039 BC00039 V=333.3 PL=0
'PRZEJAZ NAD BELKA
MOVL C00040 BC00040 V=666.7
MOVJ C00041 BC00041 VJ=40.00
MOVJ C00042 BC00042 VJ=40.00
MOVJ C00043 BC00043 VJ=40.00
'W1P
MOVJ C00044 BC00044 VJ=20.00 PL=0
MOVL C00045 BC00045 V=166.7 PL=0
REFP 3 C00046 BC00046
CALL JOB:SEARCH-R1
SET P0104 P0006
SFTON P0104
MOVL C00047 BC00047 V=166.7 PL=0
REFP 3 C00048 BC00048
CALL JOB:SEARCH-R1
SET P0104 P0006
SFTON P0104
MOVL C00049 BC00049 V=333.3 PL=0
SFTOF
'W1L
MOVL C00050 BC00050 V=666.7
MOVL C00051 BC00051 V=166.7 PL=0
REFP 3 C00052 BC00052
CALL JOB:SEARCH-R1
SET P0105 P0006
SFTON P0105
MOVL C00053 BC00053 V=166.7 PL=0
REFP 3 C00054 BC00054
CALL JOB:SEARCH-R1
SET P0105 P0006
SFTON P0105
MOVL C00055 BC00055 V=333.3 PL=0
SFTOF
MOVL C00056 BC00056 V=666.7
'W10P
MOVL C00057 BC00057 V=166.7 PL=0
REFP 3 C00058 BC00058
CALL JOB:SEARCH-R1
SET P0106 P0006
SFTON P0106
MOVL C00059 BC00059 V=166.7 PL=0
REFP 3 C00060 BC00060
CALL JOB:SEARCH-R1
SET P0106 P0006
SFTON P0106
MOVL C00061 BC00061 V=333.3 PL=0
SFTOF
'W10L
MOVL C00062 BC00062 V=333.3
MOVL C00063 BC00063 V=166.7 PL=0
REFP 3 C00064 BC00064
CALL JOB:SEARCH-R1
SET P0107 P0006
SFTON P0107
MOVL C00065 BC00065 V=166.7 PL=0
REFP 3 C00066 BC00066
CALL JOB:SEARCH-R1
SET P0107 P0006
SFTON P0107
MOVL C00067 BC00067 V=333.3 PL=0
SFTOF
MOVL C00068 BC00068 V=333.3
'PRZEJAZD
MOVJ C00069 BC00069 VJ=50.00
MOVJ C00070 BC00070 VJ=50.00
MOVJ C00071 BC00071 VJ=60.00
MOVJ C00072 BC00072 VJ=60.00
MOVJ C00073 BC00073 VJ=60.00
MOVJ C00074 BC00074 VJ=60.00 PL=0
MOVL C00075 BC00075 V=166.7 PL=0
REFP 3 C00076 BC00076
CALL JOB:SEARCH-R1
SET P0108 P0006
SFTON P0108
MOVL C00077 BC00077 V=166.7 PL=0
REFP 3 C00078 BC00078
CALL JOB:SEARCH-R1
SET P0108 P0006
SFTON P0108
MOVL C00079 BC00079 V=333.3 PL=0
SFTOF
'W2P
'W2L
MOVL C00080 BC00080 V=666.7
MOVL C00081 BC00081 V=166.7 PL=0
REFP 3 C00082 BC00082
CALL JOB:SEARCH-R1
SET P0109 P0006
SFTON P0109
MOVL C00083 BC00083 V=166.7 PL=0
REFP 3 C00084 BC00084
CALL JOB:SEARCH-R1
SET P0109 P0006
SFTON P0109
MOVL C00085 BC00085 V=333.3 PL=0
SFTOF
MOVJ C00086 BC00086 VJ=20.00
SFTOF
CALL JOB:TWIN_5340_0ST_RAMA_PRZ_OBR1_POM
'.................
'.................
'.................
'PROG POMIARY RAMA PRZED
'.................
'.................
'.................
MOVJ C00087 BC00087 VJ=50.00
'COMMENT
'COMMENT
'COMMENT
'COMMENT
'COMMENT
'COMMENT
PAUSE
COMM 'PRZEJAZD
COMM 'POMIAR DO WYJ!! PRZEROBIC NA STD
COMM 'KONIEC
COMM MOVJ C00088 BC00088 VJ=40.00
COMM MOVJ C00089 BC00089 VJ=50.00
COMM 'W5L
COMM MOVJ C00090 BC00090 VJ=30.00 PL=0
COMM SET I020 110
COMM CALL JOB:SEARCH_Z-40_Z1_X40
COMM MOVL C00091 BC00091 V=166.7
COMM 'W6L
COMM MOVJ C00092 BC00092 VJ=20.00 PL=0
COMM SET I020 112
COMM CALL JOB:SEARCH_Z-40_Z1_X40
COMM MOVL C00093 BC00093 V=166.7
COMM 'W6P
COMM MOVL C00094 BC00094 V=150.0 PL=0
COMM SET I020 113
COMM CALL JOB:SEARCH_Z-40_Z1_X40
COMM MOVL C00095 BC00095 V=166.7
COMM 'W5P
COMM MOVJ C00096 BC00096 VJ=20.00 PL=0
COMM SET I020 111
COMM CALL JOB:SEARCH_Z-40_Z1_X40
COMM MOVL C00097 BC00097 V=166.7
COMM 'W7A
COMM MOVJ C00098 BC00098 VJ=40.00
COMM MOVJ C00099 BC00099 VJ=40.00
COMM MOVJ C00100 BC00100 VJ=40.00
COMM MOVJ C00101 BC00101 VJ=40.00
COMM MOVJ C00102 BC00102 VJ=40.00
COMM MOVJ C00103 BC00103 VJ=40.00
COMM MOVJ C00104 BC00104 VJ=40.00
COMM MOVJ C00105 BC00105 VJ=40.00
COMM MOVL C00106 BC00106 V=250.0
COMM REFP 3 C00107 BC00107
COMM CALL JOB:SEARCH-R1
COMM SET P0280 P0006
COMM SFTON P0280
COMM MOVL C00108 BC00108 V=166.7
COMM MOVL C00109 BC00109 V=250.0
COMM MOVL C00110 BC00110 V=166.7
COMM REFP 3 C00111 BC00111
COMM CALL JOB:SEARCH-R1
COMM SET P0280 P0006
COMM MOVL C00112 BC00112 V=166.7
COMM SFTOF
COMM MOVL C00113 BC00113 V=333.3
COMM MOVL C00114 BC00114 V=166.7
COMM REFP 3 C00115 BC00115
COMM CALL JOB:SEARCH-R1
COMM SET P0290 P0006
COMM SFTON P0290
COMM MOVL C00116 BC00116 V=166.7
COMM REFP 3 C00117 BC00117
COMM CALL JOB:SEARCH-R1
COMM SET P0290 P0006
COMM MOVL C00118 BC00118 V=166.7
COMM 'DOKONCZYC SEARCH
COMM 'DOKONCZYC SEARCH
COMM MOVJ C00119 BC00119 VJ=20.00
COMM SFTOF
COMM MOVJ C00120 BC00120 VJ=30.00
COMM MOVJ C00121 BC00121 VJ=40.00
COMM MOVJ C00122 BC00122 VJ=40.00
COMM MOVJ C00123 BC00123 VJ=40.00
COMM MOVJ C00124 BC00124 VJ=40.00
COMM MOVJ C00125 BC00125 VJ=50.00
COMM 'W7B
COMM MOVJ C00126 BC00126 VJ=50.00
COMM MOVJ C00127 BC00127 VJ=50.00
COMM MOVJ C00128 BC00128 VJ=30.00
COMM MOVJ C00129 BC00129 VJ=20.00
COMM MOVL C00130 BC00130 V=166.7
COMM REFP 3 C00131 BC00131
COMM CALL JOB:SEARCH-R1
COMM SET P0281 P0006
COMM MOVL C00132 BC00132 V=166.7
COMM SFTON P0281
COMM MOVL C00133 BC00133 V=166.7
COMM MOVL C00134 BC00134 V=166.7
COMM REFP 3 C00135 BC00135
COMM CALL JOB:SEARCH-R1
COMM SET P0281 P0006
COMM MOVJ C00136 BC00136 VJ=15.00
COMM SFTOF
COMM MOVJ C00137 BC00137 VJ=20.00
COMM MOVL C00138 BC00138 V=166.7
COMM REFP 3 C00139 BC00139
COMM CALL JOB:SEARCH-R1
COMM SET P0291 P0006
COMM MOVL C00140 BC00140 V=166.7
COMM MOVL C00141 BC00141 V=166.7
COMM REFP 3 C00142 BC00142
COMM CALL JOB:SEARCH-R1
COMM SET P0291 P0006
COMM MOVL C00143 BC00143 V=166.7
COMM 'DOKONCZYC SEARCH
COMM 'DOKONCZYC SEARCH
COMM 'DOKONCZYC SEARCH
COMM MOVJ C00144 BC00144 VJ=30.00
COMM MOVJ C00145 BC00145 VJ=30.00
COMM MOVJ C00146 BC00146 VJ=50.00
COMM MOVJ C00147 BC00147 VJ=50.00
'------------------------
'------------------------
'PRAWA STRONA PROFIL GORA
'------------------------
'------------------------
MOVJ C00148 BC00148 VJ=50.00
MOVJ C00149 BC00149 VJ=50.00
MOVJ C00150 BC00150 VJ=50.00
MOVJ C00151 BC00151 VJ=20.00
MOVJ C00152 BC00152 VJ=50.00
'------------------------
'W14A L
'------------------------
SFTOF
MOVJ C00153 BC00153 VJ=50.00
MOVJ C00154 BC00154 VJ=30.00
MOVL C00155 BC00155 V=166.7 PL=0
REFP 3 C00156 BC00156
CALL JOB:SEARCH-R1
SET P0300 P0006
SFTON P0300
MOVL C00157 BC00157 V=166.7 PL=0
REFP 3 C00158 BC00158
CALL JOB:SEARCH-R1
SET P0300 P0006
SFTON P0300
MOVL C00159 BC00159 V=166.7 PL=0
SFTOF
'------------------------
'W14A P
'------------------------
SFTOF
MOVJ C00160 BC00160 VJ=50.00
MOVJ C00161 BC00161 VJ=50.00
MOVL C00162 BC00162 V=166.7 PL=0
REFP 3 C00163 BC00163
CALL JOB:SEARCH-R1
SET P0301 P0006
SFTON P0301
MOVL C00164 BC00164 V=166.7 PL=0
REFP 3 C00165 BC00165
CALL JOB:SEARCH-R1
SET P0301 P0006
SFTON P0301
MOVL C00166 BC00166 V=166.7 PL=0
SFTOF
'------------------------
'W19A L
'------------------------
SFTOF
MOVJ C00167 BC00167 VJ=50.00
MOVL C00168 BC00168 V=200.0 PL=0
REFP 3 C00169 BC00169
CALL JOB:SEARCH-R1
SET P0302 P0006
SFTON P0302
MOVL C00170 BC00170 V=166.7 PL=0
REFP 3 C00171 BC00171
CALL JOB:SEARCH-R1
SET P0302 P0006
SFTON P0302
MOVL C00172 BC00172 V=250.0 PL=0
SFTOF
'------------------------
'W19A P
'------------------------
SFTOF
MOVJ C00173 BC00173 VJ=50.00
MOVL C00174 BC00174 V=166.7 PL=0
REFP 3 C00175 BC00175
CALL JOB:SEARCH-R1
SET P0303 P0006
SFTON P0303
MOVL C00176 BC00176 V=166.7 PL=0
REFP 3 C00177 BC00177
CALL JOB:SEARCH-R1
SET P0303 P0006
SFTON P0303
MOVL C00178 BC00178 V=166.7 PL=0
SFTOF
'------------------------
'W13A L
'------------------------
SFTOF
MOVJ C00179 BC00179 VJ=50.00
MOVL C00180 BC00180 V=166.7 PL=0
REFP 3 C00181 BC00181
CALL JOB:SEARCH-R1
SET P0304 P0006
SFTON P0304
MOVL C00182 BC00182 V=166.7 PL=0
REFP 3 C00183 BC00183
CALL JOB:SEARCH-R1
SET P0304 P0006
SFTON P0304
MOVL C00184 BC00184 V=166.7 PL=0
SFTOF
'------------------------
'W13A P
'------------------------
SFTOF
MOVJ C00185 BC00185 VJ=50.00
MOVL C00186 BC00186 V=200.0 PL=0
REFP 3 C00187 BC00187
CALL JOB:SEARCH-R1
SET P0305 P0006
SFTON P0305
MOVL C00188 BC00188 V=166.7 PL=0
REFP 3 C00189 BC00189
CALL JOB:SEARCH-R1
SET P0305 P0006
SFTON P0305
MOVL C00190 BC00190 V=250.0 PL=0
SFTOF
'------------------------
'W18A L
'------------------------
SFTOF
MOVJ C00191 BC00191 VJ=50.00
MOVL C00192 BC00192 V=200.0 PL=0
REFP 3 C00193 BC00193
CALL JOB:SEARCH-R1
SET P0306 P0006
SFTON P0306
MOVL C00194 BC00194 V=166.7 PL=0
REFP 3 C00195 BC00195
CALL JOB:SEARCH-R1
SET P0306 P0006
SFTON P0306
MOVL C00196 BC00196 V=166.7 PL=0
SFTOF
'------------------------
'W18A P
'------------------------
SFTOF
MOVJ C00197 BC00197 VJ=50.00
MOVL C00198 BC00198 V=200.0 PL=0
REFP 3 C00199 BC00199
CALL JOB:SEARCH-R1
SET P0307 P0006
SFTON P0307
MOVL C00200 BC00200 V=166.7 PL=0
REFP 3 C00201 BC00201
CALL JOB:SEARCH-R1
SET P0307 P0006
SFTON P0307
MOVL C00202 BC00202 V=166.7 PL=0
SFTOF
'------------------------
'W15A L
'------------------------
SFTOF
MOVJ C00203 BC00203 VJ=50.00
MOVL C00204 BC00204 V=200.0 PL=0
REFP 3 C00205 BC00205
CALL JOB:SEARCH-R1
SET P0308 P0006
SFTON P0308
MOVL C00206 BC00206 V=166.7 PL=0
REFP 3 C00207 BC00207
CALL JOB:SEARCH-R1
SET P0308 P0006
SFTON P0308
MOVL C00208 BC00208 V=166.7 PL=0
SFTOF
'------------------------
'W15A P
'------------------------
SFTOF
MOVJ C00209 BC00209 VJ=50.00
MOVL C00210 BC00210 V=166.7 PL=0
REFP 3 C00211 BC00211
CALL JOB:SEARCH-R1
SET P0309 P0006
SFTON P0309
MOVL C00212 BC00212 V=166.7 PL=0
REFP 3 C00213 BC00213
CALL JOB:SEARCH-R1
SET P0309 P0006
SFTON P0309
MOVL C00214 BC00214 V=166.7 PL=0
SFTOF
MOVL C00215 BC00215 V=333.3
'------------------------
'W17A L
'------------------------
MOVL C00216 BC00216 V=500.0
SFTOF
MOVJ C00217 BC00217 VJ=20.00
MOVL C00218 BC00218 V=166.7 PL=0
REFP 3 C00219 BC00219
CALL JOB:SEARCH-R1
SET P0310 P0006
SFTON P0310
MOVL C00220 BC00220 V=166.7 PL=0
REFP 3 C00221 BC00221
CALL JOB:SEARCH-R1
SET P0310 P0006
SFTON P0310
MOVL C00222 BC00222 V=166.7 PL=0
SFTOF
'------------------------
'W17A P
'------------------------
SFTOF
MOVL C00223 BC00223 V=416.7
MOVL C00224 BC00224 V=166.7 PL=0
REFP 3 C00225 BC00225
CALL JOB:SEARCH-R1
SET P0311 P0006
SFTON P0311
MOVL C00226 BC00226 V=166.7 PL=0
REFP 3 C00227 BC00227
CALL JOB:SEARCH-R1
SET P0311 P0006
SFTON P0311
MOVL C00228 BC00228 V=166.7 PL=0
SFTOF
MOVJ C00229 BC00229 VJ=10.00
MOVJ C00230 BC00230 VJ=20.00
MOVJ C00231 BC00231 VJ=50.00
MOVJ C00232 BC00232 VJ=50.00
MOVJ C00233 BC00233 VJ=70.00
MOVJ C00234 BC00234 VJ=30.00
MOVJ C00235 BC00235 VJ=30.00
'------------------------
'------------------------
'LEWA STRONA PROFIL GORA
'------------------------
'------------------------
MOVJ C00236 BC00236 VJ=30.00
MOVJ C00237 BC00237 VJ=30.00
MOVJ C00238 BC00238 VJ=30.00
'------------------------
'W17B L
'------------------------
SFTOF
MOVJ C00239 BC00239 VJ=15.00
MOVL C00240 BC00240 V=166.7 PL=0
REFP 3 C00241 BC00241
CALL JOB:SEARCH-R1
SET P0350 P0006
SFTON P0350
MOVL C00242 BC00242 V=166.7 PL=0
REFP 3 C00243 BC00243
CALL JOB:SEARCH-R1
SET P0350 P0006
SFTON P0350
MOVL C00244 BC00244 V=166.7 PL=0
SFTOF
'------------------------
'W17B P
'------------------------
SFTOF
MOVL C00245 BC00245 V=333.3
MOVL C00246 BC00246 V=166.7 PL=0
REFP 3 C00247 BC00247
CALL JOB:SEARCH-R1
SET P0351 P0006
SFTON P0351
MOVL C00248 BC00248 V=166.7 PL=0
REFP 3 C00249 BC00249
CALL JOB:SEARCH-R1
SET P0351 P0006
SFTON P0351
MOVL C00250 BC00250 V=166.7 PL=0
SFTOF
'POPRAWID DOJAZD
'------------------------
'W15B L
'------------------------
SFTOF
MOVJ C00251 BC00251 VJ=10.00
MOVL C00252 BC00252 V=166.7 PL=0
REFP 3 C00253 BC00253
CALL JOB:SEARCH-R1
SET P0352 P0006
SFTON P0352
MOVL C00254 BC00254 V=166.7 PL=0
REFP 3 C00255 BC00255
CALL JOB:SEARCH-R1
SET P0352 P0006
SFTON P0352
MOVL C00256 BC00256 V=166.7 PL=0
SFTOF
'------------------------
'W15B P
'------------------------
SFTOF
MOVJ C00257 BC00257 VJ=20.00
MOVL C00258 BC00258 V=166.7 PL=0
REFP 3 C00259 BC00259
CALL JOB:SEARCH-R1
SET P0353 P0006
SFTON P0353
MOVL C00260 BC00260 V=166.7 PL=0
REFP 3 C00261 BC00261
CALL JOB:SEARCH-R1
SET P0353 P0006
SFTON P0353
MOVL C00262 BC00262 V=166.7 PL=0
SFTOF
'------------------------
'W18B L
'------------------------
SFTOF
MOVJ C00263 BC00263 VJ=50.00
MOVL C00264 BC00264 V=166.7 PL=0
REFP 3 C00265 BC00265
CALL JOB:SEARCH-R1
SET P0354 P0006
SFTON P0354
MOVL C00266 BC00266 V=166.7 PL=0
REFP 3 C00267 BC00267
CALL JOB:SEARCH-R1
SET P0354 P0006
SFTON P0354
MOVL C00268 BC00268 V=166.7 PL=0
SFTOF
'------------------------
'W18B P
'------------------------
SFTOF
MOVJ C00269 BC00269 VJ=50.00
MOVL C00270 BC00270 V=166.7 PL=0
REFP 3 C00271 BC00271
CALL JOB:SEARCH-R1
SET P0355 P0006
SFTON P0355
MOVL C00272 BC00272 V=166.7 PL=0
REFP 3 C00273 BC00273
CALL JOB:SEARCH-R1
SET P0355 P0006
SFTON P0355
MOVL C00274 BC00274 V=166.7 PL=0
SFTOF
'------------------------
'W13B L
'------------------------
SFTOF
MOVJ C00275 BC00275 VJ=50.00
MOVL C00276 BC00276 V=166.7 PL=0
REFP 3 C00277 BC00277
CALL JOB:SEARCH-R1
SET P0356 P0006
SFTON P0356
MOVL C00278 BC00278 V=166.7 PL=0
REFP 3 C00279 BC00279
CALL JOB:SEARCH-R1
SET P0356 P0006
SFTON P0356
MOVL C00280 BC00280 V=166.7 PL=0
SFTOF
'------------------------
'W13B P
'------------------------
SFTOF
MOVJ C00281 BC00281 VJ=50.00
MOVL C00282 BC00282 V=166.7 PL=0
REFP 3 C00283 BC00283
CALL JOB:SEARCH-R1
SET P0357 P0006
SFTON P0357
MOVL C00284 BC00284 V=166.7 PL=0
REFP 3 C00285 BC00285
CALL JOB:SEARCH-R1
SET P0357 P0006
SFTON P0357
MOVL C00286 BC00286 V=166.7 PL=0
SFTOF
'------------------------
'W19B L
'------------------------
SFTOF
MOVJ C00287 BC00287 VJ=50.00
MOVL C00288 BC00288 V=166.7 PL=0
REFP 3 C00289 BC00289
CALL JOB:SEARCH-R1
SET P0358 P0006
SFTON P0358
MOVL C00290 BC00290 V=166.7 PL=0
REFP 3 C00291 BC00291
CALL JOB:SEARCH-R1
SET P0358 P0006
SFTON P0358
MOVL C00292 BC00292 V=166.7 PL=0
SFTOF
'------------------------
'W19B P
'------------------------
SFTOF
MOVJ C00293 BC00293 VJ=50.00
MOVL C00294 BC00294 V=166.7 PL=0
REFP 3 C00295 BC00295
CALL JOB:SEARCH-R1
SET P0359 P0006
SFTON P0359
MOVL C00296 BC00296 V=166.7 PL=0
REFP 3 C00297 BC00297
CALL JOB:SEARCH-R1
SET P0359 P0006
SFTON P0359
MOVL C00298 BC00298 V=166.7 PL=0
SFTOF
'------------------------
'W14B L
'------------------------
SFTOF
MOVJ C00299 BC00299 VJ=50.00
MOVL C00300 BC00300 V=166.7 PL=0
REFP 3 C00301 BC00301
CALL JOB:SEARCH-R1
SET P0360 P0006
SFTON P0360
MOVL C00302 BC00302 V=166.7 PL=0
REFP 3 C00303 BC00303
CALL JOB:SEARCH-R1
SET P0360 P0006
SFTON P0360
MOVL C00304 BC00304 V=166.7 PL=0
SFTOF
'------------------------
'W14B P
'------------------------
SFTOF
MOVJ C00305 BC00305 VJ=50.00
MOVL C00306 BC00306 V=166.7 PL=0
REFP 3 C00307 BC00307
CALL JOB:SEARCH-R1
SET P0361 P0006
SFTON P0361
MOVL C00308 BC00308 V=166.7 PL=0
REFP 3 C00309 BC00309
CALL JOB:SEARCH-R1
SET P0361 P0006
SFTON P0361
MOVL C00310 BC00310 V=166.7 PL=0
SFTOF
MOVJ C00311 BC00311 VJ=50.00
MOVJ C00312 BC00312 VJ=50.00
MOVJ C00313 BC00313 VJ=50.00
MOVJ C00314 BC00314 VJ=50.00
'WELD
'WELD
'WELD
MOVJ C00315 BC00315 VJ=10.00
'**********************
'**********************
'POCZATEK SPAWANIA DOL
'**********************
'**********************
''
'**********************
'W1
'**********************
MOVJ C00316 BC00316 VJ=50.00
MOVJ C00317 BC00317 VJ=40.00
MOVL C00318 BC00318 V=166.7
SFTON P0104
MOVL C00319 BC00319 V=166.7
MACRO1 MJ#(0) ARGF24
ARCON
SFTON P0105
MOVL C00320 BC00320 V=11.7
ARCOF
SFTOF
MOVJ C00321 BC00321 VJ=20.00
MOVJ C00322 BC00322 VJ=30.00
MOVJ C00323 BC00323 VJ=50.00
MOVJ C00324 BC00324 VJ=40.00
MOVJ C00325 BC00325 VJ=20.00
'**********************
'W2
'**********************
SFTON P0108
MOVL C00326 BC00326 V=166.7
ARCON
SFTON P0109
MOVL C00327 BC00327 V=11.3
MOVL C00328 BC00328 V=11.3
COMM MOVL C00329 BC00329 V=11.7
ARCOF
SFTOF
MOVL C00330 BC00330 V=333.3
MOVJ C00331 BC00331 VJ=40.00
MOVJ C00332 BC00332 VJ=70.00
MOVJ C00333 BC00333 VJ=20.00
MOVL C00334 BC00334 V=666.7
'**********************
'W3
'**********************
SFTON P0101
MOVL C00335 BC00335 V=166.7
ARCON
SFTON P0100
MOVL C00336 BC00336 V=11.7
ARCOF
MOVL C00337 BC00337 V=166.7
SFTOF
MOVJ C00338 BC00338 VJ=30.00
MOVJ C00339 BC00339 VJ=30.00
MOVJ C00340 BC00340 VJ=50.00
MOVJ C00341 BC00341 VJ=30.00
MOVJ C00342 BC00342 VJ=40.00
'**********************
'W5
'**********************
MOVJ C00343 BC00343 VJ=50.00
COMM MOVJ C00344 BC00344 VJ=25.00
COMM MOVJ C00345 BC00345 VJ=30.00
'COMMENT
'COMMENT
'COMMENT
'COMMENT
CALL JOB:TWIN_5340_0ST_RAMA_PRZ_OBR1_SPAW
PAUSE
'COMMENT
'COMMENT
COMM '**********************
COMM 'W5
COMM '**********************
COMM MACRO1 MJ#(0) ARGF9
COMM SFTON P0777
COMM MOVL P0111 BP111 V=66.7
COMM ARCON
COMM MOVL P0110 BP110 V=10.0
COMM ARCOF
COMM SFTOF
COMM MOVJ C00346 BC00346 VJ=20.00
COMM MOVJ C00347 BC00347 VJ=20.00
COMM '**********************
COMM 'W6
COMM '**********************
COMM MACRO1 MJ#(0) ARGF9
COMM SFTON P0777
COMM MOVL P0113 BP113 V=66.7
COMM ARCON
COMM MOVL P0112 BP112 V=10.8
COMM ARCOF
COMM SFTOF
COMM MOVJ C00348 BC00348 VJ=10.00
COMM MOVJ C00349 BC00349 VJ=30.00
COMM MOVJ C00350 BC00350 VJ=30.00
COMM MOVJ C00351 BC00351 VJ=40.00
COMM MOVJ C00352 BC00352 VJ=40.00
COMM MOVJ C00353 BC00353 VJ=40.00
COMM MOVJ C00354 BC00354 VJ=40.00
COMM MOVJ C00355 BC00355 VJ=20.00
COMM MOVJ C00356 BC00356 VJ=10.00
COMM MOVJ C00357 BC00357 VJ=20.00
COMM MOVL C00358 BC00358 V=166.7
COMM MACRO1 MJ#(0) ARGF14
COMM MOVL C00359 BC00359 V=166.7
COMM SFTON P0280
COMM MOVL C00360 BC00360 V=166.7 PL=0
COMM ARCON ASF#(22)
COMM MOVL C00361 BC00361 V=9.2
COMM MOVL C00362 BC00362 V=9.2
COMM SFTON P0281
COMM MOVL C00363 BC00363 V=9.2
COMM MOVL C00364 BC00364 V=9.2
COMM ARCOF
COMM SFTOF
COMM MOVL C00365 BC00365 V=250.0
COMM MOVL C00366 BC00366 V=416.7
COMM MOVJ C00367 BC00367 VJ=30.00
COMM MOVJ C00368 BC00368 VJ=30.00
COMM MOVJ C00369 BC00369 VJ=30.00
COMM MOVJ C00370 BC00370 VJ=30.00
COMM MOVJ C00371 BC00371 VJ=30.00
COMM '7b
COMM MOVL C00372 BC00372 V=333.3
COMM MOVL C00373 BC00373 V=333.3
COMM SFTON P0281
COMM MOVL C00374 BC00374 V=166.7 PL=0
COMM ARCON ASF#(22)
COMM MOVL C00375 BC00375 V=9.2
COMM MOVL C00376 BC00376 V=9.2
COMM SFTON P0291
COMM MOVL C00377 BC00377 V=9.2
COMM MOVL C00378 BC00378 V=9.2
COMM MOVL C00379 BC00379 V=9.2
COMM ARCOF
COMM SFTOF
COMM 'TUTAJ DODAC 7
COMM 'TUTAJ DODAC 7
COMM 'TUTAJ DODAC 7
COMM MOVL C00380 BC00380 V=333.3
COMM MOVL C00381 BC00381 V=333.3
COMM MOVL C00382 BC00382 V=333.3
MOVJ C00383 BC00383 VJ=20.00
MOVJ C00384 BC00384 VJ=30.00
MOVJ C00385 BC00385 VJ=50.00
MOVJ C00386 BC00386 VJ=50.00
MOVJ C00387 BC00387 VJ=40.00
MOVJ C00388 BC00388 VJ=10.00
'**********************
'W9
'**********************
SFTON P0103
MACRO1 MJ#(0) ARGF24
MOVL C00389 BC00389 V=166.7 PL=0
ARCON
SFTON P0102
MOVL C00390 BC00390 V=11.7
ARCOF
SFTOF
MOVL C00391 BC00391 V=166.7
'**********************
'SPOINA_PODLOGA_BRAK_ROZP
'**********************
MOVL C00392 BC00392 V=333.3
SFTON P0099
MOVL C00393 BC00393 V=166.7
ARCON
SFTON P0098
MOVL C00394 BC00394 V=11.7
ARCOF
MOVL C00395 BC00395 V=166.7
SFTOF
'SPOINA_PODLOGA_BRAK_ROZP
MOVL C00396 BC00396 V=166.7
MOVJ C00397 BC00397 VJ=40.00
MOVJ C00398 BC00398 VJ=70.00
MOVJ C00399 BC00399 VJ=50.00
MOVJ C00400 BC00400 VJ=20.00
'**********************
'W10
'**********************
MOVL C00401 BC00401 V=333.3
SFTON P0106
MOVL C00402 BC00402 V=166.7
ARCON
SFTON P0107
MOVL C00403 BC00403 V=11.7
ARCOF
SFTOF
MOVL C00404 BC00404 V=333.3
MOVJ C00405 BC00405 VJ=50.00
'**********************
'**********************
'POCZATEK SPAWANIA BOKI
'**********************
'**********************
MOVJ C00406 BC00406 VJ=50.00
MOVJ C00407 BC00407 VJ=50.00
'**********************
'W13A
'**********************
SFTON P0305
MOVL C00408 BC00408 V=250.0 PL=0
SFTOF
MACRO1 MJ#(0) ARGF10
ARCON
SFTON P0304
MOVL C00409 BC00409 V=10.8
ARCOF
SFTOF
MOVL C00410 BC00410 V=250.0
'W13B
MOVJ C00411 BC00411 VJ=30.00
MOVJ C00412 BC00412 VJ=50.00
MOVL C00413 BC00413 V=500.0
'**********************
'W13B
'**********************
SFTON P0356
MOVL C00414 BC00414 V=133.3 PL=0
SFTOF
ARCON
SFTON P0357
MOVL C00415 BC00415 V=10.8
ARCOF
SFTOF
MOVL C00416 BC00416 V=250.0
MOVJ C00417 BC00417 VJ=30.00
MOVJ C00418 BC00418 VJ=40.00
MOVJ C00419 BC00419 VJ=30.00
MOVJ C00420 BC00420 VJ=30.00
'**********************
'W14A
'**********************
MOVL C00421 BC00421 V=250.0
SFTON P0301
MOVL C00422 BC00422 V=50.0 PL=0
SFTOF
ARCON
SFTON P0300
MOVL C00423 BC00423 V=10.8
MOVL C00424 BC00424 V=10.8
MOVL C00425 BC00425 V=10.8
ARCOF
SFTOF
MOVL C00426 BC00426 V=150.0
MOVJ C00427 BC00427 VJ=40.00
MOVJ C00428 BC00428 VJ=30.00
MOVJ C00429 BC00429 VJ=30.00
MOVJ C00430 BC00430 VJ=30.00
MOVJ C00431 BC00431 VJ=30.00
'**********************
'W14B
'**********************
SFTON P0360
MOVL C00432 BC00432 V=333.3
MOVL C00433 BC00433 V=166.7 PL=0
SFTOF
ARCON
SFTON P0361
MOVL C00434 BC00434 V=10.8
MOVL C00435 BC00435 V=10.8
MOVL C00436 BC00436 V=10.8
ARCOF
SFTOF
MOVL C00437 BC00437 V=250.0
MOVJ C00438 BC00438 VJ=40.00
MOVJ C00439 BC00439 VJ=40.00
MOVJ C00440 BC00440 VJ=30.00
MOVJ C00441 BC00441 VJ=40.00
MOVJ C00442 BC00442 VJ=30.00
MOVJ C00443 BC00443 VJ=30.00
MOVJ C00444 BC00444 VJ=30.00
MOVJ C00445 BC00445 VJ=30.00
MOVJ C00446 BC00446 VJ=30.00
'**********************
'W15A
'**********************
SFTON P0309
MOVL C00447 BC00447 V=166.7
MOVL C00448 BC00448 V=166.7 PL=0
SFTOF
ARCON
SFTON P0308
MOVL C00449 BC00449 V=10.8
ARCOF
SFTOF
MOVL C00450 BC00450 V=150.0
MOVJ C00451 BC00451 VJ=30.00
MOVJ C00452 BC00452 VJ=50.00
MOVJ C00453 BC00453 VJ=50.00
MOVJ C00454 BC00454 VJ=50.00
MOVJ C00455 BC00455 VJ=50.00
MOVJ C00456 BC00456 VJ=50.00
'**********************
'W15B
'**********************
SFTON P0352
MOVL C00457 BC00457 V=250.0
MOVL C00458 BC00458 V=83.3 PL=0
SFTOF
ARCON
SFTON P0353
MOVL C00459 BC00459 V=10.8
ARCOF
MOVL C00460 BC00460 V=166.7
SFTOF
MOVJ C00461 BC00461 VJ=40.00
MOVJ C00462 BC00462 VJ=50.00
MOVJ C00463 BC00463 VJ=50.00
'BRAK W TEJ DLUGOSCI
'**********************
'W16A
'**********************
'**********************
'W16B
'**********************
'BRAK W TEJ DLUGOSCI
'**********************
'W17A
'**********************
MOVJ C00464 BC00464 VJ=50.00
MOVJ C00465 BC00465 VJ=50.00
'**********************
'W17A
'**********************
SFTON P0310
MOVL C00466 BC00466 V=333.3
MOVL C00467 BC00467 V=166.7 PL=0
SFTOF
ARCON
SFTON P0311
MOVL C00468 BC00468 V=10.8
ARCOF
SFTOF
MOVL C00469 BC00469 V=333.3
MOVJ C00470 BC00470 VJ=30.00
MOVJ C00471 BC00471 VJ=30.00
MOVJ C00472 BC00472 VJ=50.00
MOVJ C00473 BC00473 VJ=50.00
MOVJ C00474 BC00474 VJ=50.00
MOVJ C00475 BC00475 VJ=50.00
MOVJ C00476 BC00476 VJ=50.00
MOVJ C00477 BC00477 VJ=30.00
MOVJ C00478 BC00478 VJ=30.00
'**********************
'W17B
'**********************
SFTON P0351
MOVL C00479 BC00479 V=166.7
MOVL C00480 BC00480 V=166.7 PL=0
SFTOF
ARCON
SFTON P0350
MOVL C00481 BC00481 V=10.8
ARCOF
SFTOF
MOVL C00482 BC00482 V=250.0
MOVJ C00483 BC00483 VJ=30.00
MOVJ C00484 BC00484 VJ=30.00
MOVJ C00485 BC00485 VJ=30.00
MOVJ C00486 BC00486 VJ=30.00
MOVJ C00487 BC00487 VJ=40.00
'**********************
'W18A
'**********************
SFTON P0306
MOVL C00488 BC00488 V=333.3
MOVL C00489 BC00489 V=166.7 PL=0
SFTOF
ARCON
SFTON P0307
MOVL C00490 BC00490 V=10.8
ARCOF
SFTOF
MOVL C00491 BC00491 V=250.0
MOVJ C00492 BC00492 VJ=30.00
MOVJ C00493 BC00493 VJ=30.00
MOVJ C00494 BC00494 VJ=50.00
MOVJ C00495 BC00495 VJ=50.00
MOVJ C00496 BC00496 VJ=50.00
'**********************
'W18B
'**********************
SFTON P0355
MOVL C00497 BC00497 V=166.7
MOVL C00498 BC00498 V=166.7 PL=0
SFTOF
ARCON
SFTON P0354
MOVL C00499 BC00499 V=10.8
ARCOF
MOVL C00500 BC00500 V=250.0
SFTOF
MOVJ C00501 BC00501 VJ=30.00
MOVJ C00502 BC00502 VJ=30.00
MOVJ C00503 BC00503 VJ=40.00
MOVJ C00504 BC00504 VJ=50.00
MOVJ C00505 BC00505 VJ=30.00
'**********************
'W19A
'**********************
MOVL C00506 BC00506 V=166.7
SFTON P0303
MOVL C00507 BC00507 V=166.7 PL=0
SFTOF
ARCON
SFTON P0302
MOVL C00508 BC00508 V=10.8
ARCOF
SFTOF
MOVL C00509 BC00509 V=150.0
MOVJ C00510 BC00510 VJ=30.00
MOVJ C00511 BC00511 VJ=50.00
MOVJ C00512 BC00512 VJ=50.00
'**********************
'W19B
'**********************
SFTON P0358
MOVL C00513 BC00513 V=500.0
MOVL C00514 BC00514 V=166.7 PL=0
SFTOF
ARCON
SFTON P0359
MOVL C00515 BC00515 V=10.8
ARCOF
SFTOF
MOVL C00516 BC00516 V=250.0
MOVJ C00517 BC00517 VJ=40.00
MOVJ C00518 BC00518 VJ=50.00
CALL JOB:MOVE_OUT_OF_TUNNEL
END
